TYPE EM_TransportCanSupply2_SIM :
STRUCT
END_STRUCT
END_TYPE

(* stored: Version 1.1.0.1, ProductVersion 3.1.4024.12
   DUT EM_TransportCanSupply2_SIM: Id {7454fec1-4913-41ed-8bde-f006e90fbf4f} *)
